PROGRAM Reaktoranlage
VAR
	
	MODUS			:FB_Modus;
	
	VENTIL			:FB_A_Magnetventil; 
	RUEHRER			:FB_A_Motor1R;
	PUMPE			:FB_A_Motor2R;
	HKSYSTEM		:FB_A_HKSystem;
	
	FUELLSEN		:FB_S_Fuellstandsensor;
	TEMPSEN			:FB_S_Temperatursensor; 

END_VAR

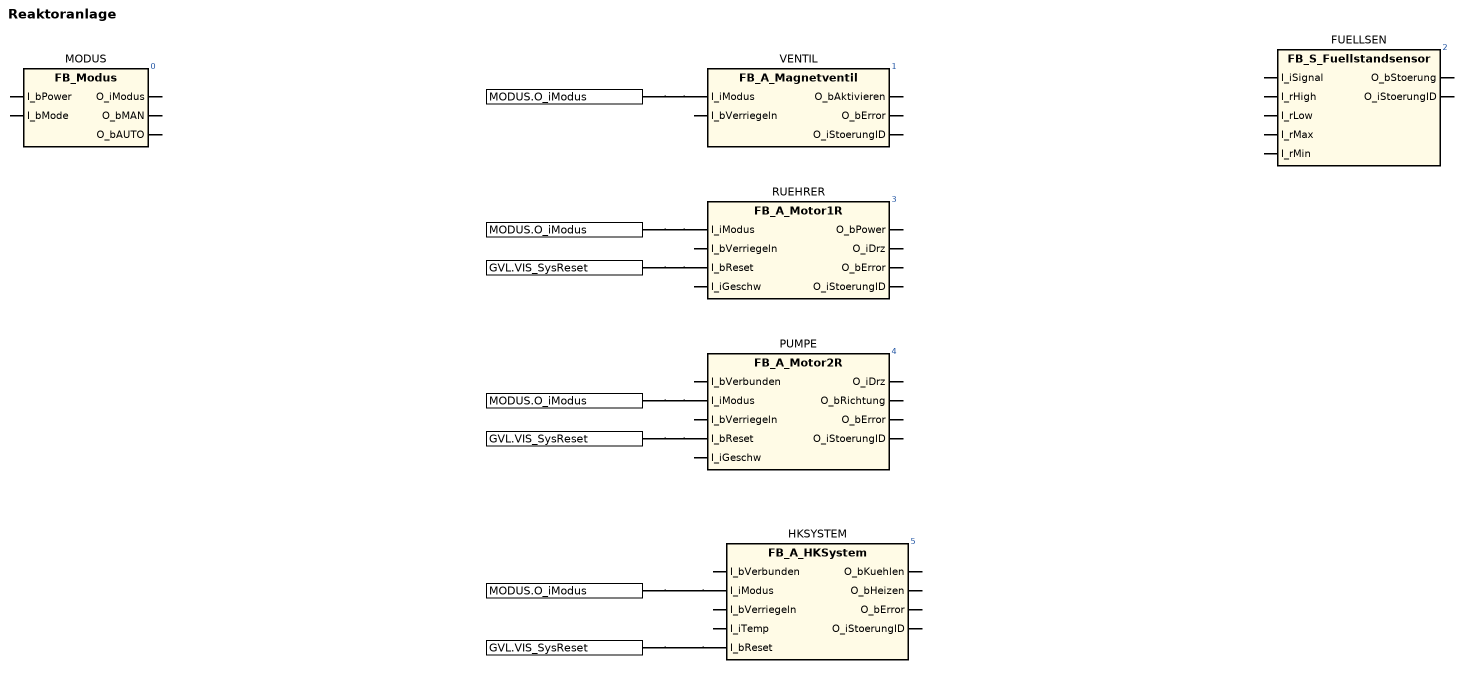
MODUS(); // FB_Modus
VENTIL(I_iModus := MODUS.O_iModus); // FB_A_Magnetventil
FUELLSEN(); // FB_S_Fuellstandsensor
RUEHRER(I_iModus := MODUS.O_iModus, I_bReset := GVL.VIS_SysReset); // FB_A_Motor1R
PUMPE(I_iModus := MODUS.O_iModus, I_bReset := GVL.VIS_SysReset); // FB_A_Motor2R
HKSYSTEM(I_iModus := MODUS.O_iModus, I_bReset := GVL.VIS_SysReset); // FB_A_HKSystem

END_PROGRAM

(* stored: Version 1.1.0.1, ProductVersion 3.1.4024.12
   POU Reaktoranlage: Id {30c67279-b6a5-4aec-833e-cd28d8c4a283}, SpecialFunc None *)
